Universal Robots URScript: Lab_exe_12_2_221.script

def Lab_exe_12_2_221():
  modbus_add_signal("172.16.17.8", 255, 0, 1, "MODBUS_1")
  modbus_set_signal_update_frequency("MODBUS_1", 10)
  modbus_add_signal("172.16.17.8", 255, 1, 1, "MODBUS_2")
  modbus_set_signal_update_frequency("MODBUS_2", 10)
  modbus_add_signal("172.16.17.8", 255, 16, 0, "MODBUS_3")
  modbus_set_signal_update_frequency("MODBUS_3", 10)
  modbus_add_signal("172.16.17.8", 255, 17, 0, "MODBUS_4")
  modbus_set_signal_update_frequency("MODBUS_4", 10)
  set_standard_analog_input_domain(0, 1)
  set_standard_analog_input_domain(1, 1)
  set_tool_analog_input_domain(0, 1)
  set_tool_analog_input_domain(1, 1)
  set_analog_outputdomain(0, 1)
  set_analog_outputdomain(1, 1)
  set_tool_voltage(24)
  set_standard_digital_input_action(0, "default")
  set_standard_digital_input_action(1, "default")
  set_standard_digital_input_action(2, "default")
  set_standard_digital_input_action(3, "default")
  set_standard_digital_input_action(4, "default")
  set_standard_digital_input_action(5, "default")
  set_standard_digital_input_action(6, "default")
  set_standard_digital_input_action(7, "default")
  set_tool_digital_input_action(0, "default")
  set_tool_digital_input_action(1, "default")
  modbus_set_runstate_dependent_choice("MODBUS_1",0)
  modbus_set_runstate_dependent_choice("MODBUS_2",0)
  set_tcp(p[0.0,0.0,0.125,0.0,0.0,0.0])
  set_payload(0.0)
  set_gravity([0.0, 0.0, 9.82])
  global i_var_1=1
  global count=1
  global select_no=1
  global force1=124.23835
  global u26426u24231=p[0.0,0.0,0.0,0.0,0.0,0.0]
  global u24037u20855=get_forward_kin()
  while (True):
    $ 1 "机器人程序"
    $ 2 "MoveJ"
    $ 3 "waypoint1"
    movej([1.5913114547729492, -1.7855525397368304, -1.865690130927275, -0.7408674399005335, 1.4744844436645508, 2.3143115043640137], a=1.3962634015954636, v=1.0471975511965976)
    $ 4 "waypoint2"
    movej([1.5913874447461809, -1.6750893580151818, -1.3285796316827714, -1.3886085501020453, 1.4726582464267963, 2.316079243170854], a=1.3962634015954636, v=1.0471975511965976)
    $ 5 "waypoint3"
    movej([1.340636818304075, -1.3555229234744246, -1.9297398202282672, -1.0943295713006433, 1.5539544441038073, 2.077707488250754], a=1.3962634015954636, v=1.0471975511965976)
  end
end
